{attribute 'GeneratedUsingTerminal: KL1212'}
{attribute addProperty BoxType "KL1212"}
{attribute addProperty Id "Channel_1AT %Q*Channel_72DF63360Channel_2AT %Q*Channel_72DF63360"}
{attribute addProperty CRC "3968136300"}
{attribute addProperty Size "0"}
TYPE KL1212_EC84F46C :
STRUCT
	{attribute addProperty Name "Channel_1"}
	Channel_1 : Channel_72DF6336;
	{attribute addProperty Name "Channel_2"}
	Channel_2 : Channel_72DF6336;
END_STRUCT
END_TYPE
